ABB RobotStudio station: mdx_20211111-163905.rsstn

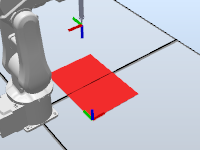
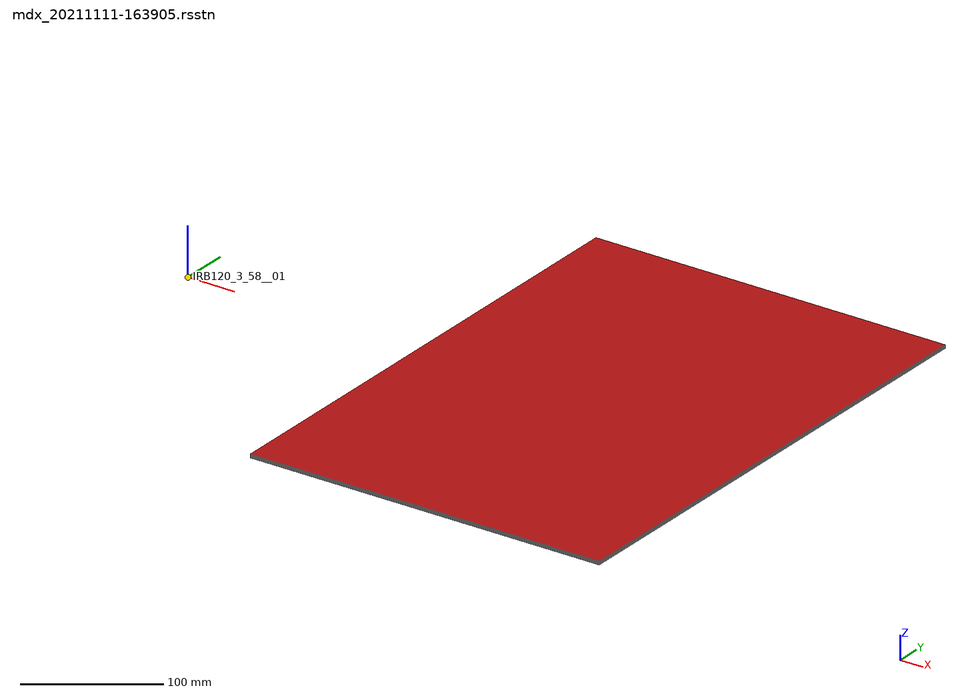
[picture v1: parts stored in the station drawn from their meshes, with robot base, taught points and paths (robot models come from the ABB library and are not in the file)]
Station mdx (saved by RobotStudio 21.2.9526.0)
Controller IRB120_3_58
  mechanical unit ROB_1: IRB120_3_58__01, 6 joints, base frame (0, 0, 0) mm
Layout (positions relative to the parent item):
  - IRB120_3_58__01 [mechanism, from Robots\IRB120_3_58_G_01.rslib] at (0, 0, 0) mm; joint values [0, 0.0001, 0, 0, 1.5708, 0] (rad or m)
  - Part_1 [part], size 297 x 420 x 3 mm
  - Group_1 [graphiccomponentgroup]
  - pen [mechanism, from Libraries\pen.rslib] at (302.02, 0, 557.98) mm, rotated rx 180 ry 0 rz 180 deg
Attachment: pen is attached to IRB120_3_58__01 / Link6
Targets, tools, work objects and paths stored in the station, written as RAPID:
! task T_ROB1
MODULE CalibData
  TASK PERS wobjdata drawing_paper:=[FALSE,TRUE,"",[[0,0,0],[1,0,0,0]],[[200.001631399,-209.998000605,3],[1,-0.000012962,0,0.000002643]]];
  PERS tooldata pen:=[TRUE,[[0,0,163.48],[1,0,0,0]],[1,[0,0,100],[1,0,0,0],0,0,0]];
ENDMODULE

! task T_ROB1
MODULE Module1
  CONST robtarget Target_10:=[[-200,200,1.5],[0,1,0,0],[0,0,0,0],[9E+09,9E+09,9E+09,9E+09,9E+09,9E+09]];
  CONST robtarget Target_20:=[[-200,210,3],[0,1,0,0],[0,0,0,0],[9E+09,9E+09,9E+09,9E+09,9E+09,9E+09]];
ENDMODULE

